// TIA Portal V17 export
// export: Created 2026-04-13T11:12:44.1115697Z, ExportSetting WithDefaults, DisplayName Totally Integrated Automation Portal, DisplayVersion V17 Update 4, DisplayName TIA Portal Openness, DisplayVersion V17 Update 4, DisplayName TIA Portal Version Control Interface, DisplayVersion V17, DisplayName SINAMICS Startdrive Advanced, DisplayVersion V17, DisplayName SINAMICS Startdrive G130, G150, S120, S150, SINAMICS MV, S210, DisplayVersion V17, DisplayName SINAMICS Startdrive G110M, G120, G120C, G120D, G120P, G115D, DisplayVersion V17, DisplayName STEP 7 Professional, DisplayVersion V17 Update 4, DisplayName STEP 7 Safety, DisplayVersion V17, DisplayName WinCC Professional, DisplayVersion V17 Update 4
FUNCTION_BLOCK "10-模拟量输入"   // FB40, SCL
{ S7_Optimized_Access := 'TRUE' }
VERSION : 0.1
// stored: AutoNumber true, IsIECCheckEnabled false, IsRetainMemResEnabled false, MemoryReserve 100, SetENOAutomatically false, UDAEnableTagReadback false
   VAR_INPUT
      HMI上限 : Real;
      HMI下限 : Real;
      PLC上限 : Int := 27648;
      PLC下限 : Int;
   END_VAR
   VAR_IN_OUT
      "PLC-仪表" : Int;
      HMI仪表 : Real;
   END_VAR
   VAR
      DBD28 : Real;
   END_VAR
BEGIN
   #DBD28 := NORM_X_REAL(MIN := #PLC下限, VALUE := #"PLC-仪表", MAX := #PLC上限);
   #HMI仪表 := SCALE_X_REAL(MIN := #HMI下限, VALUE := #DBD28, MAX := #HMI上限);
END_FUNCTION_BLOCK
